// SIMATIC STEP 7 (V5.x) project S7_m3
// CPU: CPU312(1)
// station: P_ADR_BUS
// station: Hardware
// station: SIMATIC 300 Station
// program: S7 Program(1)

SYMBOL_TABLE
"start"	I 0.0	BOOL
"stop"	I 0.1	BOOL
"reset"	I 0.2	BOOL
"pallet sensor"	I 0.3	BOOL
"box sensor"	I 0.4	BOOL
"detected"	I 0.5	BOOL
"moving X"	I 0.6	BOOL
"moving Z"	I 0.7	BOOL
"rotating"	I 1.0	BOOL
"start(light)"	Q 0.0	BOOL
"stop(light)"	Q 0.1	BOOL
"restet(light)"	Q 0.2	BOOL
"box conveyor"	Q 0.3	BOOL
"pallet conveyor"	Q 0.4	BOOL
"X"	Q 0.5	BOOL
"Z"	Q 0.6	BOOL
"rotate cw"	Q 0.7	BOOL
"rotate ccw"	Q 1.0	BOOL
"grab"	Q 1.1	BOOL
END_SYMBOL_TABLE

ORGANIZATION_BLOCK OB 1
TITLE = "Main Program Sweep (Cycle)"
VERSION : 0.1
VAR_TEMP
  OB1_EV_CLASS : BYTE ;	//Bits 0-3 = 1 (Coming event), Bits 4-7 = 1 (Event class 1)
  OB1_SCAN_1 : BYTE ;	//1 (Cold restart scan 1 of OB 1), 3 (Scan 2-n of OB 1)
  OB1_PRIORITY : BYTE ;	//Priority of OB Execution
  OB1_OB_NUMBR : BYTE ;	//1 (Organization block 1, OB1)
  OB1_RESERVED_1 : BYTE ;	//Reserved for system
  OB1_RESERVED_2 : BYTE ;	//Reserved for system
  OB1_PREV_CYCLE : INT ;	//Cycle time of previous OB1 scan (milliseconds)
  OB1_MIN_CYCLE : INT ;	//Minimum cycle time of OB1 (milliseconds)
  OB1_MAX_CYCLE : INT ;	//Maximum cycle time of OB1 (milliseconds)
  OB1_DATE_TIME : DATE_AND_TIME ;	//Date and time OB1 started
END_VAR
BEGIN
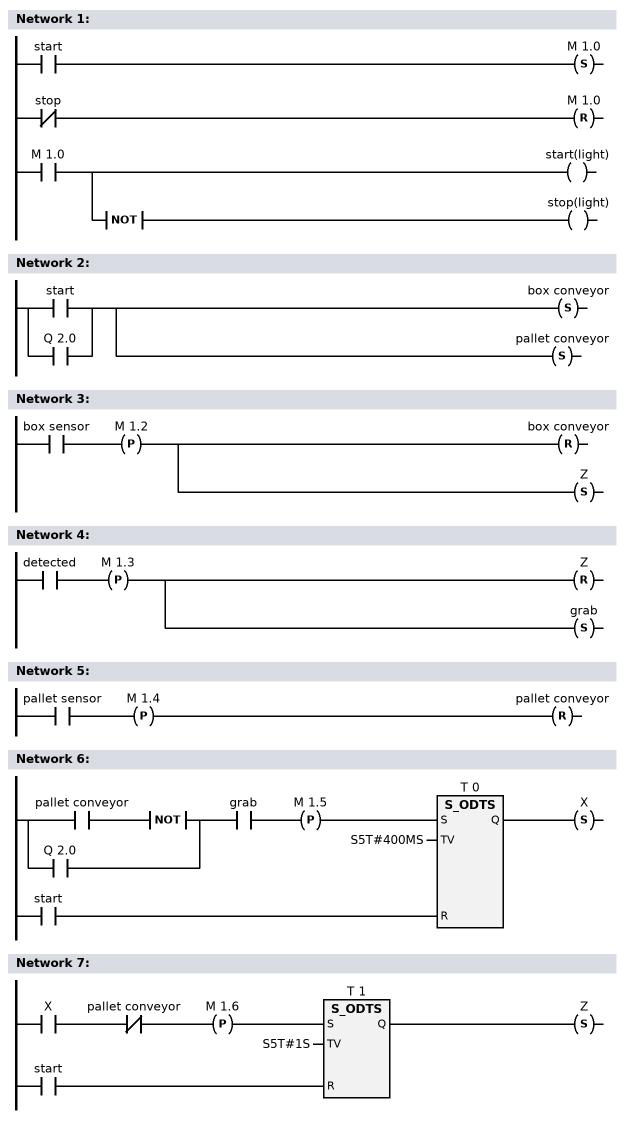
NETWORK
TITLE =
      A     "start";
      S     M 1.0;
      AN    "stop";
      R     M 1.0;
      A     M 1.0;
      =     L 20.0;
      A     L 20.0;
      BLD   102;
      =     "start(light)";
      A     L 20.0;
      NOT;
      =     "stop(light)";
NETWORK
TITLE =
      O     "start";
      O     Q 2.0;
      S     "box conveyor";
      S     "pallet conveyor";
NETWORK
TITLE =
      A     "box sensor";
      FP    M 1.2;
      R     "box conveyor";
      S     "Z";
NETWORK
TITLE =
      A     "detected";
      FP    M 1.3;
      R     "Z";
      S     "grab";
NETWORK
TITLE =
      A     "pallet sensor";
      FP    M 1.4;
      R     "pallet conveyor";
NETWORK
TITLE =
      A(;
      A     "pallet conveyor";
      NOT;
      O     Q 2.0;
      );
      A     "grab";
      FP    M 1.5;
      L     S5T#400MS;
      SS    T 0;
      A     "start";
      R     T 0;
      NOP   0;
      NOP   0;
      A     T 0;
      S     "X";
NETWORK
TITLE =
      A     "X";
      AN    "pallet conveyor";
      FP    M 1.6;
      L     S5T#1S;
      SS    T 1;
      A     "start";
      R     T 1;
      NOP   0;
      NOP   0;
      A     T 1;
      S     "Z";
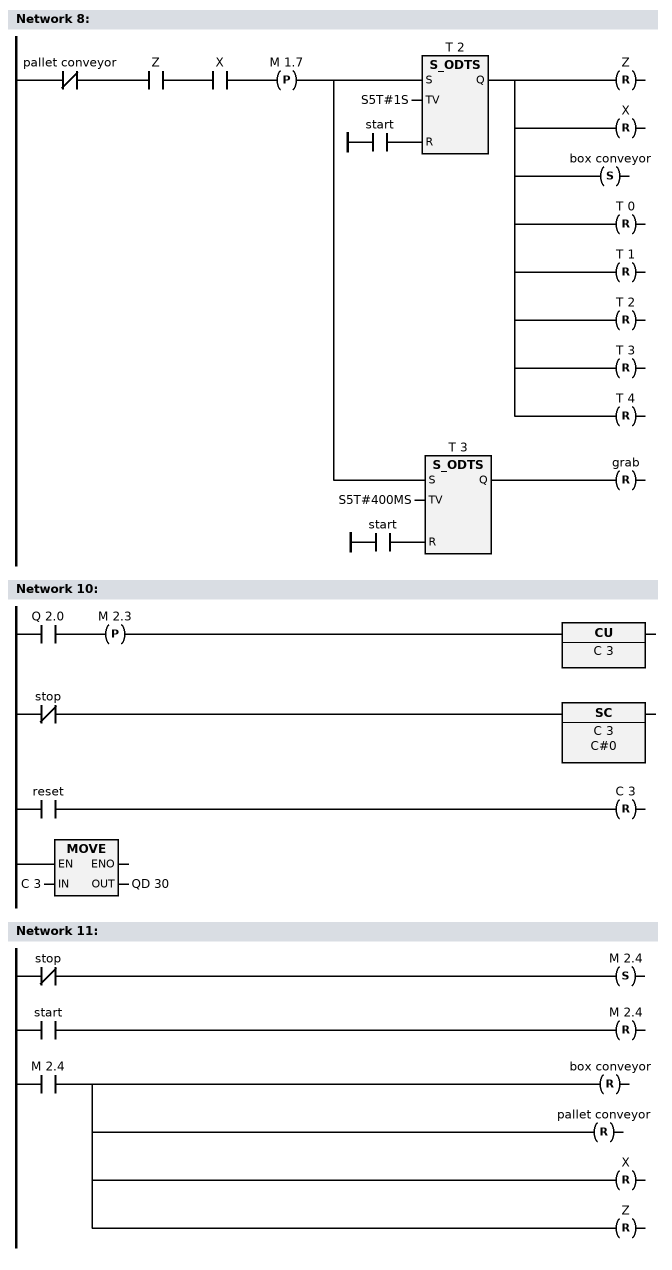
NETWORK
TITLE =
      AN    "pallet conveyor";
      A     "Z";
      A     "X";
      FP    M 1.7;
      =     L 20.0;
      A     L 20.0;
      L     S5T#1S;
      SS    T 2;
      A     "start";
      R     T 2;
      NOP   0;
      NOP   0;
      A     T 2;
      R     "Z";
      R     "X";
      S     "box conveyor";
      R     T 0;
      R     T 1;
      R     T 2;
      R     T 3;
      R     T 4;
      A     L 20.0;
      L     S5T#400MS;
      SS    T 3;
      A     "start";
      R     T 3;
      NOP   0;
      NOP   0;
      A     T 3;
      R     "grab";
NETWORK
TITLE =
      A(;
      A     "X";
      FN    M 2.2;
      CU    C 2;
      BLD   101;
      AN    "stop";
      L     C#0;
      S     C 2;
      A(;
      O     "start";
      O     Q 2.0;
      );
      R     C 2;
      L     C 2;
      T     MW 9;
      NOP   0;
      A     C 2;
      );
      A(;
      L     MW 9;
      L     2;
      ==I;
      );
      =     Q 2.0;
NETWORK
TITLE =
      A     Q 2.0;
      FP    M 2.3;
      CU    C 3;
      BLD   101;
      AN    "stop";
      L     C#0;
      S     C 3;
      A     "reset";
      R     C 3;
      L     C 3;
      T     QD 30;
      NOP   0;
      NOP   0;
NETWORK
TITLE =
      AN    "stop";
      S     M 2.4;
      A     "start";
      R     M 2.4;
      A     M 2.4;
      R     "box conveyor";
      R     "pallet conveyor";
      R     "X";
      R     "Z";
END_ORGANIZATION_BLOCK
